{attribute 'strict'}
{attribute 'to_string'}
TYPE E_MessageType :
(
  eMessageEmpty,
  eMessageInfo,
  eMessageWarn,
  eMessageError
)DINT;
END_TYPE

(* stored: Version 1.1.0.1, ProductVersion 3.1.4024.12
   DUT E_MessageType: Id {6a3c98a9-6687-0ef0-25df-25aac2ef283a} *)
